TYPE enum_E:
    (elit_loc1, elit_loc2);
END_TYPE

(* stored: ProductVersion 3.1.0.18, Version 1.1.0.1 *)
